INTERFACE ITF_BaseComplexElement_HMI_Connector EXTENDS ITF_BaseExecutiveElement_HMI_Connector

END_INTERFACE

(* stored: Version 1.1.0.1
   Itf ITF_BaseComplexElement_HMI_Connector: Id {886a85bc-d9f2-0b34-350a-7828be6ba314} *)
